(*
SPDX-FileCopyrightText: Â© 2026 Oleksandr Tiutyk <trofimich@gmail.com>
SPDX-License-Identifier: MIT
License: https://opensource.org/license/mit
*)

(*!
<summary>Represents a leaf automation component that performs cyclic input processing.</summary>
<description>
Invoked during the input phase of the component tree cycle to read physical inputs or update state.
</description>
*)

INTERFACE IInputLeafAutomationComponent EXTENDS IChildAutomationComponent

(*!
<summary>Performs cyclic reading and processing of input data.</summary>
*)
METHOD ProcessInput
END_METHOD

END_INTERFACE

(* stored: Version 1.1.0.1
   Itf IInputLeafAutomationComponent: Id {69b515a2-a927-4e6c-a8d8-6cf13a34e99e}
   Method ProcessInput: Id {067c3a3b-2632-40fe-81d7-9d2a2248bb9a} *)
